# EPICS autosave request: LabJackApp/Db/LabJackWaveformGenN_settings.req
$(P)WaveGenEnable$(N)
$(P)WaveGenType$(N)
$(P)WaveGenPulseWidth$(N)
$(P)WaveGenAmplitude$(N)
$(P)WaveGenOffset$(N)
